{attribute 'conditionalshow'}
FUNCTION_BLOCK FB_XL1XXX_DI
VAR_INPUT
	{attribute 'hide'}
	bInvers							: BOOL;				//Invert the input signal
END_VAR
VAR_OUTPUT
	{attribute 'hide'}
	bSignal							: BOOL;				//Signal from the terminal
END_VAR
VAR
	bDataIn					AT%I*	: BOOL;				//Input data from the termianl 
END_VAR

//Creator : Kai Ebensperger
//Company : Lynus AG
//Date : 02.06.2021
//Version : 1.0.0.0

//With this fuction block its possible to read in a digital signal from a Beckhoff Digital Input terminal
//Here we have the possibility to invert the input signal

IF NOT bInvers THEN 
	bSignal := bDataIn;
ELSE
	bSignal := NOT bDataIn;
END_IF

END_FUNCTION_BLOCK

(* stored: Version 1.1.0.1, ProductVersion 3.1.4024.6
   POU FB_XL1XXX_DI: Id {2fd8c04b-6e28-43e5-9831-84ea8294e675}, SpecialFunc None *)
